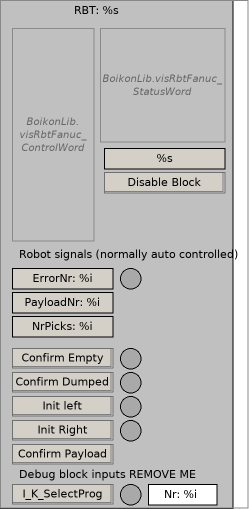
VISUALIZATION Vis_RbtFanucUnloading  // 249x509
VAR_INPUT
	I_UnitName:STRING := 'myRobot';
END_VAR

VAR_IN_OUT
	IO_cntrl: cntrl_RbtFanucUnloadingRobot;
END_VAR
    Rectangle (0,0 233x509)
    Rectangle (4,0 185x21), "RBT: %s", text variable: I_UnitName
    Frame (12,28 82x213)
        shows BoikonLib.visRbtFanuc_ControlWord(IO := IO_cntrl.DataOut.Vars._UI)
    Frame (100,28 125x114)
        shows BoikonLib.visRbtFanuc_StatusWord(IO := IO_cntrl.DataIn.Vars._UO)
    Button (104,172 121x21), "Disable Block"
        toggle IO_cntrl.TB_DisableActivations
    Ellipse (120,348 21x21), colour toggle: IO_cntrl.DataIn.Vars._DO.SN_CrateEmpty
    Button (12,348 101x20), "Confirm Empty"
        tap IO_cntrl.DataOut.Vars._DI.SN_CrateEmptyOk
    Rectangle (12,316 101x21), "NrPicks: %i", text variable: IO_cntrl.DataIn.Vars._GO.NrPickedCrates
    Button (12,372 101x20), "Confirm Dumped"
        tap IO_cntrl.DataOut.Vars._DI.SN_RequestDumpOk
    Ellipse (120,372 21x21), colour toggle: IO_cntrl.DataIn.Vars._DO.SN_RequestDump
    Ellipse (120,396 21x21), colour toggle: IO_cntrl.DataIn.Vars._DO.SN_InitLeftOk
    Ellipse (120,420 21x21), colour toggle: IO_cntrl.DataIn.Vars._DO.SN_InitRightOk
    Button (12,396 101x20), "Init left"
        toggle IO_cntrl.DataOut.Vars._DI.SN_InitLeft
    Button (12,420 101x20), "Init Right"
        toggle IO_cntrl.DataOut.Vars._DI.SN_InitRight
    Ellipse (120,268 21x21), colour toggle: IO_cntrl.DataIn.Vars._DO.STS_Error
    Rectangle (12,268 101x21), "ErrorNr: %i", text variable: IO_cntrl.DataIn.Vars._GO.ErrorNr
    Button (12,444 101x20), "Confirm Payload"
        tap IO_cntrl.DataOut.Vars._DI.SN_PayloadConfirm
    Rectangle (12,292 101x21), "PayloadNr: %i", text variable: IO_cntrl.DataIn.Vars._GO.NrPayload
    Label (16,248 233x13), "Robot signals (normally auto controlled)"
    Label (16,468 233x13), "Debug block inputs REMOVE ME"
    Button (12,484 101x20), "I_K_SelectProg"
        toggle IO_cntrl.I_K_ProgramSelect
    Ellipse (120,484 21x21), colour toggle: IO_cntrl.Q_K_ProgramSelect_OK
    Rectangle (148,484 69x21), "Nr: %i", text variable: IO_cntrl.I_SP_ProgramNr
        OnMouseClick: write the text variable via Default, min 0, max 100
    Rectangle (104,148 121x21), "%s", text variable: IO_cntrl.eS
END_VISUALIZATION

(* stored: Version 1.1.0.1
   Visu Vis_RbtFanucUnloading: Id {396f87cd-b0d5-4542-a974-100bb3ecf244} *)
